PROGRAM MAIN
VAR
END_VAR

\zx\zx

END_PROGRAM

(* stored: Version 1.1.0.1, ProductVersion 3.1.4024.5
   POU MAIN: Id {358f84d2-bc6c-4ef7-a8a1-94c01dc877a3}, SpecialFunc None *)
